{attribute 'GeneratedUsingTerminal: EK1100-0000-0018'}
{attribute addProperty BoxType "EK1100-0000-0018"}
{attribute addProperty Id "Term_147_EK1122Term_147_EK1122_CA6A5D16124Term_186_EK1122Term_186_EK1122_75C79D52124Term_148_EL1809EL1809_32157CFD20Term_149_EL1809EL1809_32157CFD20Term_150_EL1809EL1809_32157CFD20Term_151_EL1809EL1809_32157CFD20Term_152_EL1809EL1809_32157CFD20Term_288_EK1122Term_288_EK1122_18F8921F153"}
{attribute addProperty CRC "1125515021"}
{attribute addProperty Size "501"}
{attribute addProperty Name "Term 146 (EK1100)"}
TYPE Term_146_EK1100_4315FF0D EXTENDS EK1100_1FC0878B :
STRUCT
	{attribute addProperty Name "Term 147 (EK1122)"}
	{attribute addProperty PreviousPort "Term 146 (EK1100) : B"}
	{attribute addProperty SyncUnit "default"}
	Term_147_EK1122 : Term_147_EK1122_CA6A5D16;
	{attribute addProperty Name "Term 186 (EK1122)"}
	{attribute addProperty PreviousPort "Term 147 (EK1122) : C"}
	{attribute addProperty SyncUnit "default"}
	Term_186_EK1122 : Term_186_EK1122_75C79D52;
	{attribute addProperty Name "Term 148 (EL1809)"}
	{attribute addProperty PreviousPort "Term 186 (EK1122) : C"}
	{attribute addProperty SyncUnit "default"}
	Term_148_EL1809 : EL1809_32157CFD;
	{attribute addProperty Name "Term 149 (EL1809)"}
	{attribute addProperty PreviousPort "Term 148 (EL1809) : B"}
	{attribute addProperty SyncUnit "default"}
	Term_149_EL1809 : EL1809_32157CFD;
	{attribute addProperty Name "Term 150 (EL1809)"}
	{attribute addProperty PreviousPort "Term 149 (EL1809) : B"}
	{attribute addProperty SyncUnit "default"}
	Term_150_EL1809 : EL1809_32157CFD;
	{attribute addProperty Name "Term 151 (EL1809)"}
	{attribute addProperty PreviousPort "Term 150 (EL1809) : B"}
	{attribute addProperty SyncUnit "default"}
	Term_151_EL1809 : EL1809_32157CFD;
	{attribute addProperty Name "Term 152 (EL1809)"}
	{attribute addProperty PreviousPort "Term 151 (EL1809) : B"}
	{attribute addProperty SyncUnit "default"}
	Term_152_EL1809 : EL1809_32157CFD;
	{attribute addProperty Name "Term 288 (EK1122)"}
	{attribute addProperty PreviousPort "Term 152 (EL1809) : B"}
	{attribute addProperty SyncUnit "default"}
	Term_288_EK1122 : Term_288_EK1122_18F8921F;
END_STRUCT
END_TYPE

(* stored: Version 1.2.0.0, ProductVersion 3.1.4024.11
   DUT Term_146_EK1100_4315FF0D: Id {f429af2c-d604-0995-2007-3b1ce971020f} *)
